(* CODESYS project Abstract Factory1.project

Project tree, tasks and I/O mapping:
  Device : CODESYS Control for Raspberry Pi SL, 3S - Smart Software Solutions GmbH, version 3.5.11.0
    application Application
      libraries: Standard, * (System); StringUtils, 3.5.11.0 (System)
      task Task (cyclic, interval t#20ms, priority 1) calls MAIN
      function block FB_CsvLogger [ST]: Write
      function block FB_TxtLogger [ST]: Write
      function block FB_Logger [ST]: Write, FB_init, FB_exit
      function block FB_XmlLogger [ST]: Write
      interface ILogger: Write
      program MAIN [ST]
    SoftMotion General Axis Pool
    I²C
    SPI
    GPIOs_A_B : GPIOs A/B, 3S - Smart Software Solutions GmbH, version 3.5.11.0
        unmapped channels: digital inputs (GPIO0..GPIO31), digital outputs (GPIO0..GPIO31)
    Onewire
    Camera device
      <Empty>
*)

// Device/Application/MAIN
PROGRAM MAIN
VAR
	fbLogger 		: FB_Logger('File.csv');
	retMsg			: STRING;
END_VAR

(* 
The first (most obvious) step implicates developing a function block for logging or messaging. 
In the course of this, the Write() method receives the text and the function block writes the message in a text file.

Furthermore, the Write() method expands the text by the word Logger. As a check, the whole text is returned.
	
METHOD PUBLIC Write : STRING
VAR_INPUT
  sMsg    : STRING;
END_VAR
 
sMsg := CONCAT('logger: ', sMsg);
// open file
// write the message into the file
// close file
Write := sMsg;

The implementation of the function block is relatively easy.
	
PROGRAM MAIN
VAR
  fbLogger     : FB_Logger();
  sRetMsg      : STRING;
END_VAR
 
sRetMsg := fbLogger.Write('Hello');

However, if the user would like to use optionally a CSV or XML file instead of the simple text file, the developer should expand the block.
*)

retMsg := fbLogger.Write('Hello');

END_PROGRAM

// Device/Application/FB_Logger
FUNCTION_BLOCK PUBLIC FB_Logger
VAR
	pTxtLogger   : POINTER TO FB_TxtLogger;
	pCsvLogger   : POINTER TO FB_CsvLogger;
	pXmlLogger   : POINTER TO FB_XmlLogger;
	ipLogger     : ILogger;
END_VAR

METHOD PUBLIC Write : STRING
VAR_INPUT
	sMsg    : STRING;
END_VAR
IF (ipLogger <> 0) THEN
	Write := ipLogger.Write(CONCAT('logger: ', sMsg));
END_IF
END_METHOD

METHOD FB_init : BOOL
VAR_INPUT
    bInitRetains : BOOL; // if TRUE, the retain variables are initialized (warm start / cold start)
    bInCopyCode  : BOOL; // if TRUE, the instance afterwards gets moved into the copy code (online change)
    sFilename    : STRING;
END_VAR
VAR
	sFilenameExtension : STRING;
END_VAR
sFilenameExtension := RIGHT(sFilename, 3); // no more lowercase
IF (sFilenameExtension = 'txt') THEN
    pTxtLogger := __NEW(FB_TxtLogger);
    ipLogger := pTxtLogger^;
ELSIF (sFilenameExtension = 'csv') THEN
    pCsvLogger := __NEW(FB_CsvLogger);
    ipLogger := pCsvLogger^;
ELSIF (sFilenameExtension = 'xml') THEN
    pXmlLogger := __NEW(FB_XmlLogger);
    ipLogger := pXmlLogger^;
ELSE
    ipLogger := 0;
END_IF
END_METHOD

METHOD FB_exit : BOOL
VAR_INPUT
	bInCopyCode : BOOL; // if TRUE, the exit method is called for exiting an instance that is copied afterwards (online change).
END_VAR
IF (pTxtLogger <> 0) THEN
	__DELETE(pTxtLogger);
	pTxtLogger := 0;
END_IF

IF (pCsvLogger <> 0) THEN
	__DELETE(pCsvLogger);
	pCsvLogger := 0;
END_IF

IF (pXmlLogger <> 0) THEN
	__DELETE(pXmlLogger);
	pXmlLogger := 0;
END_IF
END_METHOD

END_FUNCTION_BLOCK

// Device/Application/FB_TxtLogger
{attribute 'enable_dynamic_creation'}
FUNCTION_BLOCK FB_TxtLogger IMPLEMENTS ILogger
VAR_INPUT
END_VAR
VAR_OUTPUT
END_VAR
VAR
END_VAR

METHOD PUBLIC Write : STRING
VAR_INPUT
	sMsg      : STRING;
END_VAR
Write := CONCAT('txt-', sMsg);
// open txt file
// write the message into the txt file
// close txt file
END_METHOD

END_FUNCTION_BLOCK

// Device/Application/ILogger
INTERFACE ILogger

METHOD Write : STRING
VAR_INPUT
	sMsg    : STRING;
END_VAR
END_METHOD

END_INTERFACE

// Device/Application/FB_CsvLogger
{attribute 'enable_dynamic_creation'}
FUNCTION_BLOCK FB_CsvLogger IMPLEMENTS ILogger 
VAR_INPUT
END_VAR
VAR_OUTPUT
END_VAR
VAR
END_VAR

METHOD PUBLIC Write : STRING
VAR_INPUT
	sMsg      : STRING;
END_VAR
Write := CONCAT('csv-', sMsg);
// open csv file
// write the message into the csv file
// close csv file
END_METHOD

END_FUNCTION_BLOCK

// Device/Application/FB_XmlLogger
{attribute 'enable_dynamic_creation'}
FUNCTION_BLOCK FB_XmlLogger IMPLEMENTS ILogger
VAR_INPUT
END_VAR
VAR_OUTPUT
END_VAR
VAR
END_VAR

METHOD PUBLIC Write : STRING
VAR_INPUT
	sMsg      : STRING;
END_VAR
Write := CONCAT('xml-', sMsg);
// open xml file
// write the message into the xml file
// close xml file
END_METHOD

END_FUNCTION_BLOCK
